// TIA Portal V16 export
// export: Created 2019-09-22T11:06:18.3725779Z, ExportSetting WithDefaults, DisplayName Totally Integrated Automation Portal, DisplayVersion V16, DisplayName TIA Portal Version Control Interface, DisplayVersion V16, DisplayName TIA Portal Openness, DisplayVersion V16, DisplayName STEP 7 Professional, DisplayVersion V16, DisplayName SIMATIC Energy Suite, DisplayVersion V16, DisplayName STEP 7 Safety, DisplayVersion V16, DisplayName WinCC Professional, DisplayVersion V16, DisplayName SIMATIC Visualization Architect, DisplayVersion V16
DATA_BLOCK "InstDiagStartupPlc"   // DB2002
VERSION : 0.1
// stored: AutoNumber true, InstanceOfName DiagStartupPlc, InstanceOfType FB
"DiagStartupPlc"
   // VAR_OUTPUT
   //    status : Int;
   //    instructionError : Int;
   // END_VAR
   // VAR_IN_OUT
   //    plc : "typePlc";
   // END_VAR
   // VAR
   //    statGeoAddr { ExternalAccessible := 'False'; ExternalVisible := 'False'; ExternalWritable := 'False'; S7_SetPoint := 'True'} : GEOADDR;
   //    statGeoLaddr { ExternalAccessible := 'False'; ExternalVisible := 'False'; ExternalWritable := 'False'} : HW_ANY;
   //    statActualCentralModules : USInt;
   //    statPlcModuleStates : Array[0..127] of Bool;
   // END_VAR
BEGIN
END_DATA_BLOCK
